// TwinCAT 3 PLC project HL3
// Title: High level object TwinCAT 3 library
// Company: Tomas Rompotl
// ProjectVersion: 0.0.1
// ProgramVersion: 3.1.4023.0
// libraries:
//   Tc2_Standard, * (Beckhoff Automation GmbH)
//   Tc2_System, * (Beckhoff Automation GmbH)
//   Tc2_Utilities, * (Beckhoff Automation GmbH)
//   Tc3_Module, * (Beckhoff Automation GmbH)
//   Base Interfaces,newest,System
// project tree:
//   DataProcessing/Comparison/ CompareAnyType.TcPOU, ComparisonTest.TcPOU, IsGreaterThanOrEqualAnyType.TcPOU, IsNotEqualAnyType.TcPOU, IsLessThanOrEqualAnyType.TcPOU, IsLessThanAnyType.TcPOU, IsEqualAnyType.TcPOU, E_Compare.TcDUT, IsGreaterThanAnyType.TcPOU
//   DataProcessing/QuickSort/ Partition.TcPOU, QuickSort.TcPOU, QuickSortTest.TcPOU
//   DataProcessing/Sort/ E_Order.TcTLEO, SortTest.TcPOU, ST_TestStruct.TcDUT, ST_TestStruct2.TcDUT, _Partition.TcPOU, _QuickSort.TcPOU, Sort.TcPOU
//   General/ E_GeneralResult.TcDUT, E_GeneralStatus.TcTLEO, NegateGeneralResult.TcPOU, Swap.TcPOU, SwapByAddr.TcPOU
//   Lists/ListOfINT/ ListOfINT.TcPOU, ListOfINTTest.TcPOU, NodeINT.TcDUT
//   Lists/List/ List.TcPOU, ListTest.TcPOU, Node.TcDUT
//   Lists/WrappableList/ExampleWithUserDatatype/ WrappableListExample.TcPOU, ListOfUserDatatype.TcPOU, UserDatatype.TcDUT
//   Lists/WrappableList/ WrappableList.TcPOU
//   Misc/ GetAnyType.TcPOU
//   / PlcTask.TcTTO
//   POUs/ MAIN.TcPOU
//   Stringify/ AnyTypeToWSTRING.TcPOU, AnyTypeToSTRING.TcPOU, Stringify.TcPOU
// real-time tasks:
//   TASK PlcTask: cycle T#10ms, priority 20, ADS port 350

CONFIGURATION HL3
    RESOURCE PLC ON TwinCAT3
        TASK PlcTask(INTERVAL := T#10ms, PRIORITY := 20);
        PROGRAM MAIN WITH PlcTask : MAIN;
    END_RESOURCE
END_CONFIGURATION

// ---- DataProcessing/Comparison/E_Compare.TcDUT

{attribute 'qualified_only'}
{attribute 'strict'}
TYPE E_Compare :
(
	EQUAL,
	NOT_EQUAL,
	LESS_THAN,
	LOWER_THAN_OR_EQUAL,
	GREATER_THAN,
	GREATER_THAN_OR_EQUAL
);
END_TYPE

// ---- DataProcessing/Sort/E_Order.TcTLEO

{attribute 'qualified_only'}
{attribute 'strict'}
TYPE E_Order :
(
	ASCENDING,
	DESCENDING
);
END_TYPE

// ---- DataProcessing/Sort/ST_TestStruct.TcDUT
TYPE ST_TestStruct :
STRUCT
	by_this	: ST_TestStruct2;
END_STRUCT
END_TYPE

// ---- DataProcessing/Sort/ST_TestStruct2.TcDUT
TYPE ST_TestStruct2 :
STRUCT
	nested_variable : TIME;
END_STRUCT
END_TYPE

// ---- General/E_GeneralResult.TcDUT

{attribute 'qualified_only'}
{attribute 'strict'}
TYPE E_GeneralResult :
(
	NONE := 0,
	OK,
	NOK,
	_TRUE, // TRUE is keyword
	_FALSE // FALSE is keyword
	
);
END_TYPE

// ---- General/E_GeneralStatus.TcTLEO

{attribute 'qualified_only'}
{attribute 'strict'}
TYPE E_GeneralStatus :
(
	NONE := 0,
	STOP,
	BUSY,
	DONE,
	ERROR,
	INPUT_ERROR,
	INTERRUPT
);
END_TYPE

// ---- Lists/ListOfINT/NodeINT.TcDUT
{attribute 'enable_dynamic_creation'}
TYPE NodeINT :
STRUCT
	data : INT;
	next : POINTER TO NodeINT;
END_STRUCT
END_TYPE

// ---- Lists/List/Node.TcDUT

{attribute 'enable_dynamic_creation'}
TYPE Node :
STRUCT
	data : POINTER TO BYTE;
	next : POINTER TO Node;
END_STRUCT
END_TYPE

// ---- Lists/WrappableList/ExampleWithUserDatatype/UserDatatype.TcDUT
TYPE UserDatatype :
STRUCT
	VarBOOL : BOOL;
	VarREAL : REAL;
	VarARRAYINT : ARRAY[0..9] OF INT;
END_STRUCT
END_TYPE

// ---- POUs/MAIN.TcPOU

PROGRAM MAIN
VAR
	a : ARRAY[0..5] OF REAL;
	b : ARRAY[10..15] OF REAL;
END_VAR


ListOfINTTest();
ListTest();
WrappableListExample();

QuickSortTest();
SortTest();
ComparisonTest();

END_PROGRAM

// ---- Lists/ListOfINT/ListOfINTTest.TcPOU
PROGRAM ListOfINTTest
VAR
	listOfINTExample : ListOfINT;
	
	// init
	first : BOOL := TRUE;
	reinit : BOOL;
	
	// insert test
	insertTest : BOOL;
	insertNumber : INT := 42;
	insertIndex : INT := 0;
	
	// remove test
	removeTest : BOOL;
	removeIndex : INT := 0;
	
	// prepend test
	prependTest : BOOL;
	prependData : INT := -10;
	
	// removeAll test
	removeAllTest : BOOL;
	
	// debug
	test : ARRAY[0..30] OF INT;
	
	// hokusy pokusy
	info : __SYSTEM.VAR_INFO;
	
END_VAR

IF first THEN
	first := FALSE;
	listOfINTExample.Append(3);
	listOfINTExample.Append(4);
	listOfINTExample.Append(5).Prepend(2).Prepend(1);
END_IF;
IF reinit THEN
	reinit := FALSE;
	listOfINTExample.FB_init(FALSE, FALSE);
	first := TRUE;
END_IF

IF insertTest THEN
	insertTest := FALSE;
	listOfINTExample.Insert(insertIndex, insertNumber);
END_IF
IF removeTest THEN
	removeTest := FALSE;
	listOfINTExample.Remove(removeIndex);
END_IF
IF removeAllTest THEN
	removeAllTest := FALSE;
	listOfINTExample.RemoveAll();
END_IF


info := __VARINFO(listOfINTExample);
test[0] := listOfINTExample.Get(0);
test[1] := listOfINTExample.Get(1);
test[2] := listOfINTExample.Get(2);
test[3] := listOfINTExample.Get(3);
test[4] := listOfINTExample.Get(4);
test[5] := listOfINTExample.Get(5);
test[6] := listOfINTExample.Get(6);
test[7] := listOfINTExample.Get(7);
test[8] := listOfINTExample.Get(8);
test[9] := listOfINTExample.Get(9);

test[20] := listOfINTExample.Get(-1);
test[21] := listOfINTExample.Get(-2);
test[22] := listOfINTExample.Get(-3);
test[23] := listOfINTExample.Get(-4);
test[24] := listOfINTExample.Get(-5);
test[25] := listOfINTExample.Get(-6);
test[26] := listOfINTExample.Get(-7);
test[27] := listOfINTExample.Get(-8);
test[28] := listOfINTExample.Get(-9);
test[29] := listOfINTExample.Get(-10);

listOfINTExample.count;

END_PROGRAM

// ---- Lists/ListOfINT/ListOfINT.TcPOU

FUNCTION_BLOCK ListOfINT
VAR_INPUT
END_VAR
VAR_OUTPUT
	count : UINT;
END_VAR
VAR
	head : POINTER TO NodeINT := NULL;
	tail : POINTER TO NodeINT := NULL;
END_VAR


// linked list implementation reference:
// https://www.codesdope.com/blog/article/c-linked-lists-in-c-singly-linked-list/


METHOD Append : REFERENCE TO ListOfINT
VAR_INPUT
	data : INT;
END_VAR
VAR
	new : POINTER TO NodeINT;
END_VAR

Append REF= THIS^;

new := __NEW(NodeINT);
new^.data := data;
new^.next := NULL;

IF head = NULL THEN
	head := new;
	tail := new;
ELSE
	tail^.next := new;
	tail := tail^.next;
END_IF
count := count + 1;
END_METHOD


METHOD Get : INT
VAR_INPUT
	// indexing from end allowed
	// index = 0 returns first element
	// index = 1 returns seconds element
	// index = -1 returns last element
	// index = -2 return before-last element
	index : INT;
END_VAR
VAR
	current : POINTER TO NodeINT := NULL;
	getIndex : INT;
	i : INT;
END_VAR

IF head = NULL THEN
	Get := 0;
	RETURN;
END_IF;

// Calculate actual index in List
getIndex := (count * BOOL_TO_INT(index < 0)) + index;

// Return 0 for invalid indexes
IF 	(getIndex >= count) OR	// Indexing from begin begins with 0
	(getIndex < 0) // Indexing from end begins with -1
THEN
	Get := 0;
	RETURN;
END_IF


current := head;
FOR i := 1 TO getIndex DO // we already got head in previous line, that's why it's from 1
	IF current^.next = NULL THEN
		Get := 0; RETURN;
	END_IF
	current := current^.next;
END_FOR
Get := current^.data;
END_METHOD

// Inserts new element into given index. Negative indexing is supported
METHOD Insert : REFERENCE TO ListOfINT
VAR_INPUT
	(*
		0 = Prepend;
		1 = Insert into second position;
		-2 = Insert into second position from end;
		-1 = Append;
	*)
	index : INT;
	data : INT;
END_VAR
VAR
	new : POINTER TO NodeINT;
	current : POINTER TO NodeINT;
	insertIndex : INT;
	i : INT;
END_VAR

Insert REF= THIS^;

new := __NEW(NodeINT);
new^.data := data;

// Calculate actual index in List
insertIndex := ((count + 1) * BOOL_TO_INT(index < 0)) + index;

IF insertIndex >= count // Index too high -> append to end
THEN
	Append(data);
	RETURN;
ELSIF insertIndex <= 0 // Index too high from the end -> prepend to beginning
THEN
	Prepend(data);
	RETURN;
END_IF

current := head;
FOR i := 1 TO insertIndex - 1 DO
	current := current^.next;
END_FOR
new^.next := current^.next;
current^.next := new;
count := count + 1;
END_METHOD


METHOD IsEmpty : BOOL
VAR_INPUT
END_VAR

IsEmpty := head = NULL;
END_METHOD


// Pushes data to the beginning of the list
METHOD Prepend : REFERENCE TO ListOfINT
VAR_INPUT
	data : INT;
END_VAR
VAR
	new : POINTER TO NodeINT;
END_VAR

Prepend REF= THIS^;

new := __NEW(NodeINT);
new^.data := data;
new^.next := head;

IF head = NULL THEN
	head := new;
	tail := new;
ELSE
	head := new;
END_IF
count := count + 1;
END_METHOD


METHOD Remove : REFERENCE TO ListOfINT;
VAR_INPUT
	index : INT;
END_VAR
VAR
	current : POINTER TO NodeINT := NULL;
	removeIndex : INT;	
	nodeToRemove : POINTER TO NodeINT;
	i : INT;
END_VAR

Remove REF= THIS^;

IF head = NULL THEN
	RETURN;
END_IF;

// Calculate actual index in List
removeIndex := (count * BOOL_TO_INT(index < 0)) + index; 

// Cancel removal for invalid indexes
IF 	(removeIndex >= count) OR // Indexing from begin begins with 0
	(removeIndex < 0) // Indexing from end begins with -1
THEN
	RETURN;
END_IF

IF removeIndex = 0 THEN
	nodeToRemove := head;
	head := head^.next;
ELSE
	current := head;
	FOR i := 1 TO removeIndex - 1 DO
		current := current^.next;
	END_FOR
	nodeToRemove := current^.next;
	current^.next := current^.next^.next;
END_IF
IF nodeToRemove = tail THEN
	tail := current;
END_IF
__DELETE(nodeToRemove);
count := count - 1;
END_METHOD


METHOD RemoveAll : REFERENCE TO ListOfINT
VAR_INPUT
END_VAR

WHILE head <> NULL DO
	Remove(0);
END_WHILE
END_METHOD

END_FUNCTION_BLOCK

// ---- Lists/List/ListTest.TcPOU

PROGRAM ListTest
VAR
	//testing
	testList : List;
	testVar	: REAL;
	appendTest : BOOL := TRUE;
	getTest : BOOL := TRUE;
	removeTest : BOOL;
	getVar : ARRAY[0..19] OF REAL;
	
END_VAR


IF appendTest THEN
	appendTest := FALSE;
	testVar := 1;
	testList.Append(testVar);
	testVar := 2;
	testList.Append(testVar);
	testVar := 3.14;
	testList.Append(testVar);
	testVar := -2;
	testList.Prepend(testVar);
	testVar := -3;
	testList.Prepend(testVar);
	testVar := -1;
	testList.Insert(2, testVar);
	testVar := 3;
	testList.Insert(5, testVar);
END_IF
IF getTest THEN
//	getTest := FALSE;
	ClearTestReadArray();
	testList.Get(0, getVar[0]);
	testList.Get(1, getVar[1]);
	testList.Get(2, getVar[2]);
	testList.Get(3, getVar[3]);
	testList.Get(4, getVar[4]);
	testList.Get(5, getVar[5]);
	testList.Get(6, getVar[6]);
	testList.Get(7, getVar[7]);
	testList.Get(8, getVar[8]);
	
	testList.Get(-1, getVar[10]);
	testList.Get(-2, getVar[11]);
	testList.Get(-3, getVar[12]);
	testList.Get(-4, getVar[13]);
	testList.Get(-5, getVar[14]);
	testList.Get(-6, getVar[15]);
	testList.Get(-7, getVar[16]);
	testList.Get(-8, getVar[17]);
END_IF
IF removeTest THEN
	removeTest := FALSE;
	testList.Remove(1);
END_IF

METHOD ClearTestReadArray : BOOL
VAR
	i : INT;
END_VAR
FOR i := 0 TO 19 DO
	getVar[i] := 0;
END_FOR
END_METHOD

END_PROGRAM

// ---- Lists/List/List.TcPOU

FUNCTION_BLOCK List
VAR_INPUT
END_VAR
VAR_OUTPUT
	count : UINT;
	_typeClass : __SYSTEM.TYPE_CLASS; // Type of data object - primitives or Userdef
	_classSize : DINT; // Size of data object - useful to check type of Userdef typeclass
END_VAR
VAR
	head : POINTER TO Node := NULL;
	tail : POINTER TO Node := NULL;
END_VAR


METHOD Append : REFERENCE TO List
VAR_INPUT
	data : ANY;
END_VAR
VAR
	new : POINTER TO Node;
END_VAR

Append REF= THIS^;

IF NOT IsTypeClassCorrect(data) THEN
	RETURN;
END_IF
SetTypeClass(data);

new := __NEW(Node);
new^.data := __NEW(BYTE, classSize);
MEMCPY(new^.data, data.pValue, classSize);
new^.next := NULL;

IF head = NULL THEN
	head := new;
	tail := new;
ELSE
	tail^.next := new;
	tail := tail^.next;
END_IF
count := count + 1;
END_METHOD


//{attribute 'monitoring' := 'call'}
// Size of data object - useful to check type of Userdef typeclass
PROPERTY classSize : DINT
GET

classSize := _classSize;
END_GET
SET // PRIVATE

_classSize := classSize;
END_SET
END_PROPERTY


METHOD Get : REFERENCE TO List
VAR_INPUT
	// indexing from end allowed
	// index = 0 returns first element
	// index = 1 returns seconds element
	// index = -1 returns last element
	// index = -2 return before-last element
	index : INT;
	destinationVariable : ANY;
END_VAR
VAR
	current : POINTER TO Node := NULL;
	getIndex : INT;
	i : INT;
END_VAR

IF NOT IsTypeClassCorrect(destinationVariable) THEN
	RETURN;
END_IF;

IF head = NULL THEN
	RETURN;
END_IF;

// Calculate actual index in List
getIndex := (count * BOOL_TO_INT(index < 0)) + index;

// Return 0 for invalid indexes
IF 	(getIndex >= count) OR	// Indexing from begin begins with 0
	(getIndex < 0) // Indexing from end begins with -1
THEN
	RETURN;
END_IF


current := head;
FOR i := 1 TO getIndex DO // we already got head in previous line, that's why it's from 1
	IF current^.next = NULL THEN
		RETURN;
	END_IF
	current := current^.next;
END_FOR
MEMMOVE(destinationVariable.pValue, current^.data, classSize);
END_METHOD

// Inserts new element into given index. Negative indexing is supported
METHOD Insert : REFERENCE TO List
VAR_INPUT
	(*
		0 = Prepend;
		1 = Insert into second position;
		-2 = Insert into second position from end;
		-1 = Append;
	*)
	index : INT;
	data : ANY;
END_VAR
VAR
	new : POINTER TO Node;
	current : POINTER TO Node;
	insertIndex : INT;
	i : INT;
END_VAR

Insert REF= THIS^;

IF NOT IsTypeClassCorrect(data) THEN
	RETURN;
END_IF
SetTypeClass(data);

new := __NEW(Node);
new^.data := __NEW(BYTE, classSize);
MEMCPY(new^.data, data.pValue, classSize);

// Calculate actual index in List
insertIndex := ((count + 1) * BOOL_TO_INT(index < 0)) + index;

IF insertIndex >= count // Index too high -> append to end
THEN
	Append(data);
	RETURN;
ELSIF insertIndex <= 0 // Index too high from the end -> prepend to beginning
THEN
	Prepend(data);
	RETURN;
END_IF

current := head;
FOR i := 1 TO insertIndex - 1 DO
	current := current^.next;
END_FOR
new^.next := current^.next;
current^.next := new;
count := count + 1;
END_METHOD


METHOD IsEmpty : BOOL
VAR_INPUT
END_VAR

IsEmpty := head = NULL;
END_METHOD


METHOD IsTypeClassCorrect : BOOL
VAR_INPUT
	CheckedVariable : ANY;
END_VAR

IF classSize = 0 THEN
	IsTypeClassCorrect := TRUE;
	RETURN;
END_IF
IsTypeClassCorrect := typeClass = CheckedVariable.TypeClass AND classSize = CheckedVariable.diSize;
END_METHOD


// Pushes data to the beginning of the list
METHOD Prepend : REFERENCE TO List
VAR_INPUT
	data : ANY;
END_VAR
VAR
	new : POINTER TO Node;
END_VAR

Prepend REF= THIS^;

IF NOT IsTypeClassCorrect(data) THEN
	RETURN;
END_IF
SetTypeClass(data);

new := __NEW(Node);
new^.data := __NEW(BYTE, classSize);
MEMCPY(new^.data, data.pValue, classSize);
new^.next := head;

IF head = NULL THEN
	head := new;
	tail := new;
ELSE
	head := new;
END_IF
count := count + 1;
END_METHOD


METHOD Remove : REFERENCE TO List;
VAR_INPUT
	index : INT;
END_VAR
VAR
	current : POINTER TO Node := NULL;
	removeIndex : INT;	
	nodeToRemove : POINTER TO Node;
	i : INT;
END_VAR

Remove REF= THIS^;

IF head = NULL THEN
	RETURN;
END_IF;

// Calculate actual index in List
removeIndex := (count * BOOL_TO_INT(index < 0)) + index; 

// Cancel removal for invalid indexes
IF 	(removeIndex >= count) OR // Indexing from begin begins with 0
	(removeIndex < 0) // Indexing from end begins with -1
THEN
	RETURN;
END_IF

IF removeIndex = 0 THEN
	nodeToRemove := head;
	head := head^.next;
ELSE
	current := head;
	FOR i := 1 TO removeIndex - 1 DO
		current := current^.next;
	END_FOR
	nodeToRemove := current^.next;
	current^.next := current^.next^.next;
END_IF
IF nodeToRemove = tail THEN
	tail := current;
END_IF
__DELETE(nodeToRemove^.data);
__DELETE(nodeToRemove);
count := count - 1;
END_METHOD


METHOD RemoveAll : REFERENCE TO List
VAR_INPUT
END_VAR

WHILE head <> NULL DO
	Remove(0);
END_WHILE
END_METHOD


METHOD SetTypeClass : BOOL
VAR_INPUT
	ReferenceVariable : ANY; // Pass any variable of your chosen type. It will only be used to obtain data type
END_VAR

IF classSize = 0 THEN
	typeClass := ReferenceVariable.TypeClass;
	classSize := ReferenceVariable.diSize;
	SetTypeClass := TRUE;
END_IF
END_METHOD


//{attribute 'monitoring' := 'call'}
// Type of data object - primitives or Userdef
PROPERTY typeClass : __SYSTEM.TYPE_CLASS
GET

typeClass := _typeClass;
END_GET
SET // PRIVATE

_typeClass := typeClass;
END_SET
END_PROPERTY

END_FUNCTION_BLOCK

// ---- Lists/WrappableList/ExampleWithUserDatatype/WrappableListExample.TcPOU
PROGRAM WrappableListExample
VAR
	myList	: ListOfUserDatatype;
	
	data1 : UserDatatype;
	data2 : UserDatatype;
	
	dataRead : UserDatatype;
	boolRead : BOOL;
	boolTest : BOOL;
	append : BOOL := TRUE;
	
	
END_VAR

IF append THEN
	data1.VarBOOL := TRUE;
	data1.VarREAL := 3.14;
	data1.VarARRAYINT[0] := 1;
	data1.VarARRAYINT[1] := 2;
	data1.VarARRAYINT[2] := 4;
	data1.VarARRAYINT[3] := -8;
	data1.VarARRAYINT[4] := -16;
	
	data2.VarBOOL := FALSE;
	data2.VarREAL := 1.618;
	data2.VarARRAYINT[0] := -555;
	data2.VarARRAYINT[1] := 123;
	data2.VarARRAYINT[2] := -10;
	data2.VarARRAYINT[3] := -0;
	data2.VarARRAYINT[4] := -18;

	append := FALSE;
	myList.Append(data1).Append(data2);
END_IF

myList.Get(0);

boolRead := myList.Get(0).VarBOOL;
myList.Get(0).VarREAL;

dataRead := myList.Get(1);

END_PROGRAM

// ---- Lists/WrappableList/ExampleWithUserDatatype/ListOfUserDatatype.TcPOU
FUNCTION_BLOCK ListOfUserDatatype EXTENDS WrappableList
VAR_INPUT
END_VAR
VAR_OUTPUT
END_VAR
VAR
END_VAR

METHOD Append : REFERENCE TO ListOfUserDatatype
VAR_INPUT
	data : UserDatatype;
END_VAR
Append REF= THIS^;
SUPER^._Append(data);
END_METHOD


METHOD Get : REFERENCE TO UserDatatype
VAR_INPUT
	index : INT;
END_VAR
VAR
	value : UserDatatype;
END_VAR

_Get(index, value);
Get REF= value;
END_METHOD

END_FUNCTION_BLOCK

// ---- Lists/WrappableList/WrappableList.TcPOU

FUNCTION_BLOCK WrappableList
VAR_INPUT
END_VAR
VAR_OUTPUT
	count : UINT;
	_typeClass : __SYSTEM.TYPE_CLASS; // Type of data object - primitives or Userdef
	_classSize : DINT; // Size of data object - useful to check type of Userdef typeclass
END_VAR
VAR
	head : POINTER TO Node := NULL;
	tail : POINTER TO Node := NULL;
END_VAR

METHOD PROTECTED _Append : REFERENCE TO WrappableList
VAR_INPUT
	data : ANY;
END_VAR
VAR
	new : POINTER TO Node;
END_VAR
_Append REF= THIS^;

IF NOT IsTypeClassCorrect(data) THEN
	RETURN;
END_IF
SetTypeClass(data);

new := __NEW(Node);
new^.data := __NEW(BYTE, classSize);
MEMCPY(new^.data, data.pValue, classSize);
new^.next := NULL;

IF head = NULL THEN
	head := new;
	tail := new;
ELSE
	tail^.next := new;
	tail := tail^.next;
END_IF
count := count + 1;
END_METHOD


METHOD PROTECTED _Get : REFERENCE TO WrappableList
VAR_INPUT
	// indexing from end allowed
	// index = 0 returns first element
	// index = 1 returns seconds element
	// index = -1 returns last element
	// index = -2 return before-last element
	index : INT;
	destinationVariable : ANY;
END_VAR
VAR
	current : POINTER TO Node := NULL;
	getIndex : INT;
	i : INT;
END_VAR

IF NOT IsTypeClassCorrect(destinationVariable) THEN
	RETURN;
END_IF;

IF head = NULL THEN
	RETURN;
END_IF;

// Calculate actual index in List
getIndex := (count * BOOL_TO_INT(index < 0)) + index;

// Return 0 for invalid indexes
IF 	(getIndex >= count) OR	// Indexing from begin begins with 0
	(getIndex < 0) // Indexing from end begins with -1
THEN
	RETURN;
END_IF


current := head;
FOR i := 1 TO getIndex DO // we already got head in previous line, that's why it's from 1
	IF current^.next = NULL THEN
		RETURN;
	END_IF
	current := current^.next;
END_FOR
MEMMOVE(destinationVariable.pValue, current^.data, classSize);
END_METHOD


//{attribute 'monitoring' := 'call'}
// Size of data object - useful to check type of Userdef typeclass
PROPERTY classSize : DINT
GET

classSize := _classSize;
END_GET
SET // PRIVATE

_classSize := classSize;
END_SET
END_PROPERTY

// Inserts new element into given index. Negative indexing is supported
METHOD Insert : REFERENCE TO WrappableList
VAR_INPUT
	(*
		0 = Prepend;
		1 = Insert into second position;
		-2 = Insert into second position from end;
		-1 = Append;
	*)
	index : INT;
	data : ANY;
END_VAR
VAR
	new : POINTER TO Node;
	current : POINTER TO Node;
	insertIndex : INT;
	i : INT;
END_VAR

Insert REF= THIS^;

IF NOT IsTypeClassCorrect(data) THEN
	RETURN;
END_IF
SetTypeClass(data);

new := __NEW(Node);
new^.data := __NEW(BYTE, classSize);
MEMCPY(new^.data, data.pValue, classSize);

// Calculate actual index in List
insertIndex := ((count + 1) * BOOL_TO_INT(index < 0)) + index;

IF insertIndex >= count // Index too high -> append to end
THEN
	_Append(data);
	RETURN;
ELSIF insertIndex <= 0 // Index too high from the end -> prepend to beginning
THEN
	Prepend(data);
	RETURN;
END_IF

current := head;
FOR i := 1 TO insertIndex - 1 DO
	current := current^.next;
END_FOR
new^.next := current^.next;
current^.next := new;
count := count + 1;
END_METHOD


METHOD IsEmpty : BOOL
VAR_INPUT
END_VAR

IsEmpty := head = NULL;
END_METHOD


METHOD IsTypeClassCorrect : BOOL
VAR_INPUT
	CheckedVariable : ANY;
END_VAR

IF classSize = 0 THEN
	IsTypeClassCorrect := TRUE;
	RETURN;
END_IF
IsTypeClassCorrect := typeClass = CheckedVariable.TypeClass AND classSize = CheckedVariable.diSize;
END_METHOD


// Pushes data to the beginning of the list
METHOD Prepend : REFERENCE TO WrappableList
VAR_INPUT
	data : ANY;
END_VAR
VAR
	new : POINTER TO Node;
END_VAR

Prepend REF= THIS^;

IF NOT IsTypeClassCorrect(data) THEN
	RETURN;
END_IF
SetTypeClass(data);

new := __NEW(Node);
new^.data := __NEW(BYTE, classSize);
MEMCPY(new^.data, data.pValue, classSize);
new^.next := head;

IF head = NULL THEN
	head := new;
	tail := new;
ELSE
	head := new;
END_IF
count := count + 1;
END_METHOD


METHOD Remove : REFERENCE TO WrappableList;
VAR_INPUT
	index : INT;
END_VAR
VAR
	current : POINTER TO Node := NULL;
	removeIndex : INT;	
	nodeToRemove : POINTER TO Node;
	i : INT;
END_VAR

Remove REF= THIS^;

IF head = NULL THEN
	RETURN;
END_IF;

// Calculate actual index in List
removeIndex := (count * BOOL_TO_INT(index < 0)) + index; 

// Cancel removal for invalid indexes
IF 	(removeIndex >= count) OR // Indexing from begin begins with 0
	(removeIndex < 0) // Indexing from end begins with -1
THEN
	RETURN;
END_IF

IF removeIndex = 0 THEN
	nodeToRemove := head;
	head := head^.next;
ELSE
	current := head;
	FOR i := 1 TO removeIndex - 1 DO
		current := current^.next;
	END_FOR
	nodeToRemove := current^.next;
	current^.next := current^.next^.next;
END_IF
IF nodeToRemove = tail THEN
	tail := current;
END_IF
__DELETE(nodeToRemove^.data);
__DELETE(nodeToRemove);
count := count - 1;
END_METHOD


METHOD RemoveAll : REFERENCE TO WrappableList
VAR_INPUT
END_VAR

WHILE head <> NULL DO
	Remove(0);
END_WHILE
END_METHOD


METHOD SetTypeClass : BOOL
VAR_INPUT
	ReferenceVariable : ANY; // Pass any variable of your chosen type. It will only be used to obtain data type
END_VAR

IF classSize = 0 THEN
	typeClass := ReferenceVariable.TypeClass;
	classSize := ReferenceVariable.diSize;
	SetTypeClass := TRUE;
END_IF
END_METHOD


//{attribute 'monitoring' := 'call'}
// Type of data object - primitives or Userdef
PROPERTY typeClass : __SYSTEM.TYPE_CLASS
GET

typeClass := _typeClass;
END_GET
SET // PRIVATE

_typeClass := typeClass;
END_SET
END_PROPERTY

END_FUNCTION_BLOCK

// ---- DataProcessing/QuickSort/QuickSortTest.TcPOU

PROGRAM QuickSortTest
VAR
	TestArray0 : ARRAY[0..20] OF REAL := [
		1, 2, 3, 4, 5, 6, 7, 8, 9, 10,
		42, 3.14, 0.618, 1.618, 2.618
	];
	TestArray1 : ARRAY[0..1] OF REAL := [0.1, -0.2];
	
	init : BOOL;
	sort : BOOL;
END_VAR


IF init THEN
	init := FALSE;
	reinit();
END_IF

IF sort THEN
	sort := FALSE;
	QuickSort(TestArray0, 0, 20);
	QuickSort(TestArray1, 0, 1);
END_IF


METHOD reinit : BOOL
VAR_INPUT
END_VAR
VAR CONSTANT
	Array0 : ARRAY[0..20] OF REAL := [
		1, 2, 3, 4, 5, 6, 7, 8, 9, 10,
		42, 3.14, 0.618, 1.618, 2.618
	];
	Array1 : ARRAY[0..1] OF REAL := [0.1, -0.2];
END_VAR

TestArray0 := Array0;
TestArray1 := Array1;
END_METHOD

END_PROGRAM

// ---- DataProcessing/Sort/Sort.TcPOU

// sort any array of anything
FUNCTION Sort : E_GeneralStatus
VAR_INPUT
	Arr 			: ANY; // data to be sorted, get size of array
	FirstElement 	: ANY; // get size of element to be able to get count of elements and iterate over them
	SortBy 			: ANY; // possibility to pass array of structures and sort by some of its member - this will get its type and offset in element. Will have its own function SortBy() later
	Order 			: E_Order;
END_VAR
VAR
	ElemSize		: DINT;
	ElemCount 		: DINT;
	MemberOffset 	: DWORD;
	
	StartIndex 		: DINT := 0;
	EndIndex 		: DINT;
END_VAR


IF 	arr.pValue = 0 OR firstElement.pValue = 0 OR sortBy.pValue = 0 OR 
	arr.diSize = 0 OR firstElement.diSize = 0 OR sortBy.pValue = 0 THEN

	Sort := E_GeneralStatus.INPUT_ERROR;
	RETURN;
END_IF

elemCount := arr.diSize / firstElement.diSize;
memberOffset := sortBy.pValue - firstElement.pValue;
EndIndex := ElemCount - 1;

_QuickSort(Arr, FirstElement, SortBy, MemberOffset, StartIndex, EndIndex, Order);

END_FUNCTION

// ---- DataProcessing/Sort/_QuickSort.TcPOU

FUNCTION _QuickSort
VAR_INPUT
	Arr					: __SYSTEM.AnyType;
	FirstElement		: __SYSTEM.AnyType;
	SortBy				: __SYSTEM.AnyType;
	MemberOffset		: DWORD;
	StartIndex			: DINT; // Start index
	EndIndex			: DINT; // End index
	Order 				: E_Order;
END_VAR
VAR 
	PivotIndex			: DINT; // Partitioning point
END_VAR


IF StartIndex < EndIndex THEN

	PivotIndex := _Partition(Arr, FirstElement, SortBy, MemberOffset, StartIndex, EndIndex, Order);
	_QuickSort(Arr, FirstElement, SortBy, MemberOffset, StartIndex, PivotIndex - 1, Order);
	_QuickSort(Arr, FirstElement, SortBy, MemberOffset, PivotIndex + 1, EndIndex, Order);
END_IF

END_FUNCTION

// ---- DataProcessing/Sort/_Partition.TcPOU

// Function used in QuickSort
FUNCTION _Partition : DINT
VAR_INPUT
	Arr					: __SYSTEM.AnyType;
	FirstElement		: __SYSTEM.AnyType;
	SortBy				: __SYSTEM.AnyType;
	MemberOffset		: DWORD;
	StartIndex			: DINT; // Starting comparision index
	EndIndex			: DINT; // Ending comparision index
	Order 				: E_Order;
END_VAR
VAR
	Pivot				: POINTER TO BYTE; // Compared number
	Leftwall			: DINT; // New pivot location
	Iterator			: DINT; // For iterator variable
	IterAdr				: POINTER TO BYTE;
	compA				: __SYSTEM.AnyType := SortBy; // get data of compared variable
	compB				: __SYSTEM.AnyType := SortBy;
END_VAR


Pivot := Arr.pValue + FirstElement.diSize * EndIndex;

Leftwall := StartIndex;

FOR Iterator := StartIndex TO EndIndex - 1 DO

	IterAdr := Arr.pValue + FirstElement.diSize * Iterator;
	
	compA.pValue := IterAdr + MemberOffset; // data of compared variable stays the same, just point to other value
	compB.pValue := Pivot + MemberOffset;
	
	CASE Order OF
		E_Order.ASCENDING:
			IF IsLessThanOrEqualAnyType(compA, compB) = E_GeneralResult._TRUE THEN

				SwapByAddr(IterAdr, Arr.pValue + FirstElement.diSize * Leftwall, FirstElement.diSize);
				Leftwall := Leftwall + 1;
			END_IF
		E_Order.DESCENDING:
			IF IsGreaterThanOrEqualAnyType(compA, compB) = E_GeneralResult._TRUE THEN

				SwapByAddr(IterAdr, Arr.pValue + FirstElement.diSize * Leftwall, FirstElement.diSize);
				Leftwall := Leftwall + 1;
			END_IF
	END_CASE
END_FOR

SwapByAddr(Arr.pValue + FirstElement.diSize * Leftwall, Pivot, FirstElement.diSize);

_Partition := Leftwall;

END_FUNCTION

// ---- DataProcessing/Comparison/IsLessThanOrEqualAnyType.TcPOU
FUNCTION IsLessThanOrEqualAnyType : E_GeneralResult
VAR_INPUT
	A					: __SYSTEM.AnyType; // A and B have to be same type
	B					: __SYSTEM.AnyType; // A and B have to be same type
END_VAR

IsLessThanOrEqualAnyType := NegateGeneralResult(IsGreaterthanAnyType(A, B));

END_FUNCTION

// ---- General/NegateGeneralResult.TcPOU

FUNCTION NegateGeneralResult : E_GeneralResult
VAR_INPUT
	result		: E_GeneralResult;
END_VAR
VAR
END_VAR


CASE result OF
	E_GeneralResult.OK:
		NegateGeneralResult := E_GeneralResult.NOK;
	E_GeneralResult.NOK:
		NegateGeneralResult := E_GeneralResult.OK;
	E_GeneralResult._TRUE:
		NegateGeneralResult := E_GeneralResult._FALSE;
	E_GeneralResult._FALSE:
		NegateGeneralResult := E_GeneralResult._TRUE;
	ELSE
		NegateGeneralResult := result;
END_CASE

END_FUNCTION

// ---- DataProcessing/Comparison/IsGreaterThanAnyType.TcPOU

FUNCTION IsGreaterThanAnyType : E_GeneralResult
VAR_INPUT
	A					: __SYSTEM.AnyType; // A and B have to be same type
	B					: __SYSTEM.AnyType; // A and B have to be same type
END_VAR
VAR
	isGreaterThan			: BOOL;
END_VAR


IF A.TypeClass <> B.TypeClass THEN

	RETURN;
END_IF

CASE UDINT_TO_INT(A.TypeClass) OF
    IBaseLibrary.TypeClass.TYPE_BOOL :
        isGreaterThan := PBOOL_TO_BOOL(a.pValue) > PBOOL_TO_BOOL(b.pValue);
    IBaseLibrary.TypeClass.TYPE_BIT :
        isGreaterThan := BYTE_TO_BIT(a.pValue^) > BYTE_TO_BIT(b.pValue^);
    IBaseLibrary.TypeClass.TYPE_BYTE :
        isGreaterThan := a.pValue^ > b.pValue^;
    IBaseLibrary.TypeClass.TYPE_WORD :
        isGreaterThan := PWORD_TO_WORD(a.pValue) > PWORD_TO_WORD(b.pValue);
    IBaseLibrary.TypeClass.TYPE_DWORD :
        isGreaterThan := PDWORD_TO_DWORD(a.pValue) > PDWORD_TO_DWORD(b.pValue);
    IBaseLibrary.TypeClass.TYPE_LWORD :
        isGreaterThan := PLWORD_TO_LWORD(a.pValue) > PLWORD_TO_LWORD(b.pValue);
    IBaseLibrary.TypeClass.TYPE_SINT :
        isGreaterThan := PSINT_TO_SINT(a.pValue) > PSINT_TO_SINT(b.pValue);
    IBaseLibrary.TypeClass.TYPE_INT :
        isGreaterThan := PINT_TO_INT(a.pValue) > PINT_TO_INT(b.pValue);
    IBaseLibrary.TypeClass.TYPE_DINT :
        isGreaterThan := PDINT_TO_DINT(a.pValue) > PDINT_TO_DINT(b.pValue);
    IBaseLibrary.TypeClass.TYPE_LINT :
        isGreaterThan := PLINT_TO_LINT(a.pValue) > PLINT_TO_LINT(b.pValue);
    IBaseLibrary.TypeClass.TYPE_USINT :
        isGreaterThan := PUSINT_TO_USINT(a.pValue) > PUSINT_TO_USINT(b.pValue);
    IBaseLibrary.TypeClass.TYPE_UINT :
        isGreaterThan := PUINT_TO_UINT(a.pValue) > PUINT_TO_UINT(b.pValue);
    IBaseLibrary.TypeClass.TYPE_UDINT :
        isGreaterThan := PUDINT_TO_UDINT(a.pValue) > PUDINT_TO_UDINT(b.pValue);
    IBaseLibrary.TypeClass.TYPE_ULINT :
        isGreaterThan := PULINT_TO_ULINT(a.pValue) > PULINT_TO_ULINT(b.pValue);
    IBaseLibrary.TypeClass.TYPE_REAL :
        isGreaterThan := PREAL_TO_REAL(a.pValue) > PREAL_TO_REAL(b.pValue);
    IBaseLibrary.TypeClass.TYPE_LREAL :
        isGreaterThan := PLREAL_TO_LREAL(a.pValue) > PLREAL_TO_LREAL(b.pValue);
    IBaseLibrary.TypeClass.TYPE_STRING :
        isGreaterThan := PSTRING_TO_STRING(a.pValue) > PSTRING_TO_STRING(b.pValue);
    IBaseLibrary.TypeClass.TYPE_TIME :
        isGreaterThan := PTIME_TO_TIME(a.pValue) > PTIME_TO_TIME(b.pValue);
    IBaseLibrary.TypeClass.TYPE_DATE :
        isGreaterThan := PDATE_TO_DATE(a.pValue) > PDATE_TO_DATE(b.pValue);
    IBaseLibrary.TypeClass.TYPE_DATEANDTIME :
        isGreaterThan := PDT_TO_DT(a.pValue) > PDT_TO_DT(b.pValue);
    IBaseLibrary.TypeClass.TYPE_TIMEOFDAY :
        isGreaterThan := PTOD_TO_TOD(a.pValue) > PTOD_TO_TOD(b.pValue);
    IBaseLibrary.TypeClass.TYPE_POINTER :
        isGreaterThan := a.pValue > b.pValue;
    IBaseLibrary.TypeClass.TYPE_LTIME :
        isGreaterThan := PLTIME_TO_LTIME(a.pValue) > PLTIME_TO_LTIME(b.pValue);
	ELSE
		RETURN;
END_CASE

IF isGreaterThan THEN

	IsGreaterThanAnyType := E_GeneralResult._TRUE;
ELSE

	IsGreaterThanAnyType := E_GeneralResult._FALSE;
END_IF

END_FUNCTION

// ---- General/SwapByAddr.TcPOU

// Swaps values of to variables
FUNCTION SwapByAddr : E_GeneralStatus
VAR_INPUT
	A : POINTER TO BYTE;
	B : POINTER TO BYTE;
	Length : DINT;
END_VAR
VAR
	Temp : POINTER TO BYTE;
END_VAR


IF A = 0 OR B = 0 THEN
	
	SwapByAddr := E_GeneralStatus.INPUT_ERROR;
	RETURN;
END_IF

Temp := __NEW(BYTE, Length);

MEMCPY(Temp, A, Length);
MEMCPY(A, B, Length);
MEMCPY(B, Temp, Length);

__DELETE(Temp);

SwapByAddr := E_GeneralStatus.DONE;

END_FUNCTION

// ---- DataProcessing/Comparison/IsGreaterThanOrEqualAnyType.TcPOU
FUNCTION IsGreaterThanOrEqualAnyType : E_GeneralResult
VAR_INPUT
	A					: __SYSTEM.AnyType; // A and B have to be same type
	B					: __SYSTEM.AnyType; // A and B have to be same type
END_VAR

IsGreaterThanOrEqualAnyType := NegateGeneralResult(IsLessThanAnyType(A, B));

END_FUNCTION

// ---- DataProcessing/Comparison/IsLessThanAnyType.TcPOU
FUNCTION IsLessThanAnyType : E_GeneralResult
VAR_INPUT
	A					: __SYSTEM.AnyType; // A and B have to be same type
	B					: __SYSTEM.AnyType; // A and B have to be same type
END_VAR
VAR
	isLessThan			: BOOL;
END_VAR

IF A.TypeClass <> B.TypeClass THEN

	RETURN;
END_IF

CASE UDINT_TO_INT(A.TypeClass) OF
    IBaseLibrary.TypeClass.TYPE_BOOL :
        isLessThan := PBOOL_TO_BOOL(a.pValue) < PBOOL_TO_BOOL(b.pValue);
    IBaseLibrary.TypeClass.TYPE_BIT :
        isLessThan := BYTE_TO_BIT(a.pValue^) < BYTE_TO_BIT(b.pValue^);
    IBaseLibrary.TypeClass.TYPE_BYTE :
        isLessThan := a.pValue^ < b.pValue^;
    IBaseLibrary.TypeClass.TYPE_WORD :
        isLessThan := PWORD_TO_WORD(a.pValue) < PWORD_TO_WORD(b.pValue);
    IBaseLibrary.TypeClass.TYPE_DWORD :
        isLessThan := PDWORD_TO_DWORD(a.pValue) < PDWORD_TO_DWORD(b.pValue);
    IBaseLibrary.TypeClass.TYPE_LWORD :
        isLessThan := PLWORD_TO_LWORD(a.pValue) < PLWORD_TO_LWORD(b.pValue);
    IBaseLibrary.TypeClass.TYPE_SINT :
        isLessThan := PSINT_TO_SINT(a.pValue) < PSINT_TO_SINT(b.pValue);
    IBaseLibrary.TypeClass.TYPE_INT :
        isLessThan := PINT_TO_INT(a.pValue) < PINT_TO_INT(b.pValue);
    IBaseLibrary.TypeClass.TYPE_DINT :
        isLessThan := PDINT_TO_DINT(a.pValue) < PDINT_TO_DINT(b.pValue);
    IBaseLibrary.TypeClass.TYPE_LINT :
        isLessThan := PLINT_TO_LINT(a.pValue) < PLINT_TO_LINT(b.pValue);
    IBaseLibrary.TypeClass.TYPE_USINT :
        isLessThan := PUSINT_TO_USINT(a.pValue) < PUSINT_TO_USINT(b.pValue);
    IBaseLibrary.TypeClass.TYPE_UINT :
        isLessThan := PUINT_TO_UINT(a.pValue) < PUINT_TO_UINT(b.pValue);
    IBaseLibrary.TypeClass.TYPE_UDINT :
        isLessThan := PUDINT_TO_UDINT(a.pValue) < PUDINT_TO_UDINT(b.pValue);
    IBaseLibrary.TypeClass.TYPE_ULINT :
        isLessThan := PULINT_TO_ULINT(a.pValue) < PULINT_TO_ULINT(b.pValue);
    IBaseLibrary.TypeClass.TYPE_REAL :
        isLessThan := PREAL_TO_REAL(a.pValue) < PREAL_TO_REAL(b.pValue);
    IBaseLibrary.TypeClass.TYPE_LREAL :
        isLessThan := PLREAL_TO_LREAL(a.pValue) < PLREAL_TO_LREAL(b.pValue);
    IBaseLibrary.TypeClass.TYPE_STRING :
        isLessThan := PSTRING_TO_STRING(a.pValue) < PSTRING_TO_STRING(b.pValue);
    IBaseLibrary.TypeClass.TYPE_TIME :
        isLessThan := PTIME_TO_TIME(a.pValue) < PTIME_TO_TIME(b.pValue);
    IBaseLibrary.TypeClass.TYPE_DATE :
        isLessThan := PDATE_TO_DATE(a.pValue) < PDATE_TO_DATE(b.pValue);
    IBaseLibrary.TypeClass.TYPE_DATEANDTIME :
        isLessThan := PDT_TO_DT(a.pValue) < PDT_TO_DT(b.pValue);
    IBaseLibrary.TypeClass.TYPE_TIMEOFDAY :
        isLessThan := PTOD_TO_TOD(a.pValue) < PTOD_TO_TOD(b.pValue);
    IBaseLibrary.TypeClass.TYPE_POINTER :
        isLessThan := a.pValue < b.pValue;
    IBaseLibrary.TypeClass.TYPE_LTIME :
        isLessThan := PLTIME_TO_LTIME(a.pValue) < PLTIME_TO_LTIME(b.pValue);
	ELSE
		RETURN;
END_CASE

IF isLessThan THEN

	IsLessThanAnyType := E_GeneralResult._TRUE;
ELSE

	IsLessThanAnyType := E_GeneralResult._FALSE;
END_IF

END_FUNCTION

// ---- DataProcessing/QuickSort/QuickSort.TcPOU

// Will sort array of REAL using QuickSort algorithm
FUNCTION QuickSort
VAR_IN_OUT
	ArrayOfREALToSort	: ARRAY[*] OF REAL; // Array to sort
END_VAR
VAR_INPUT
	FirstIndex			: INT; // Start index
	LastIndex			: INT; // End index
END_VAR
VAR 
	PivotLocation		: INT; // Partitioning point
END_VAR


IF FirstIndex < LastIndex THEN
	PivotLocation := Partition(ArrayOfREALToSort, FirstIndex, LastIndex);
	QuickSort(ArrayOfREALToSort, FirstIndex, PivotLocation - 1);
	QuickSort(ArrayOfREALToSort, PivotLocation + 1, LastIndex);
END_IF

END_FUNCTION

// ---- DataProcessing/QuickSort/Partition.TcPOU

// Function used in QuickSort
FUNCTION Partition : INT
VAR_IN_OUT
	ArrayOfREAL			: ARRAY[*] OF REAL; // Partition this array from index nLow to index nHigh
END_VAR
VAR_INPUT
	FirstIndex			: INT; // Starting comparision index
	LastIndex			: INT; // Ending comparision index
END_VAR
VAR
	Pivot				: REAL; // Compared number
	Leftwall			: INT; // New pivot location
	Iterator			: INT; // For iterator variable
END_VAR


Pivot := ArrayOfREAL[LastIndex];
Leftwall := FirstIndex;

FOR Iterator := FirstIndex TO LastIndex - 1 DO
	IF ArrayOfREAL[Iterator] <= Pivot THEN
		Swap(ArrayOfREAL[Iterator], ArrayOfREAL[Leftwall]);
		Leftwall := Leftwall + 1;
	END_IF
END_FOR

Swap(ArrayOfREAL[Leftwall], ArrayOfREAL[LastIndex]);

Partition := Leftwall;

END_FUNCTION

// ---- General/Swap.TcPOU

// Swaps values of to variables
FUNCTION Swap : E_GeneralStatus
VAR_INPUT
	A : ANY;
	B : ANY;
END_VAR
VAR
	Temp : POINTER TO BYTE;
END_VAR


IF a.pValue = 0 OR b.pValue = 0 OR a.diSize <> b.diSize THEN
	
	Swap := E_GeneralStatus.INPUT_ERROR;
	RETURN;
END_IF

Temp := __NEW(BYTE, A.diSize);

MEMCPY(Temp, A.pValue, A.diSize);
MEMCPY(A.pValue, B.pValue, A.diSize);
MEMCPY(B.pValue, Temp, A.diSize);

__DELETE(Temp);

Swap := E_GeneralStatus.DONE;

END_FUNCTION

// ---- DataProcessing/Sort/SortTest.TcPOU

PROGRAM SortTest
VAR
	TestArray0 : ARRAY[0..20] OF REAL := [
		1, 2, 3, 4, 5, 6, 7, 8, 9, 10,
		42, 3.14, 0.618, 1.618, 2.618
	];
	TestArray1 : ARRAY[0..3] OF STRING := ['aaa', 'g', 'aab', 'a'];
	
	sort_array : ARRAY[0..3] OF ST_TestStruct;	// TestArray2
	
	init : BOOL := TRUE;
	startSort : BOOL;
	
	order	: E_Order;
END_VAR


IF init THEN

	init := FALSE;

	reinit();
END_IF

IF startSort THEN

	startSort := FALSE;

	Sort(TestArray0, TestArray0[0], TestArray0[0], order);
	Sort(TestArray1, TestArray1[0], TestArray1[0], order);

	Sort(sort_array, sort_array[0], sort_array[0].by_this.nested_variable, order);
END_IF


METHOD reinit : BOOL
VAR_INPUT
END_VAR
VAR CONSTANT
	Array0 : ARRAY[0..20] OF REAL := [
		1, 2, 3, 4, 5, 6, 7, 8, 9, 10,
		42, 3.14, 0.618, 1.618, 2.618
	];
	Array1 : ARRAY[0..3] OF STRING := ['aaa', 'g', 'aab', 'a'];
END_VAR

TestArray0 := Array0;
TestArray1 := Array1;

sort_array[0].by_this.nested_variable := T#5S;
sort_array[1].by_this.nested_variable := T#1S;
sort_array[2].by_this.nested_variable := T#18D;
sort_array[3].by_this.nested_variable := T#42MS;
END_METHOD

END_PROGRAM

// ---- DataProcessing/Comparison/ComparisonTest.TcPOU
PROGRAM ComparisonTest
VAR
	r1 : LREAL := 3.14;
	r2 : LREAL := -129;
	s1 : STRING := 'towel';
	s2 : STRING := 'galaxy';
	
	at1 : __SYSTEM.AnyType;
	at2 : __SYSTEM.AnyType;
	
	res_r : ARRAY[0..6] OF E_GeneralResult;
	res_s : ARRAY[0..6] OF E_GeneralResult;
	
	test : BOOL;
	
	
	
END_VAR

IF test THEN

	test := FALSE;

	at1 := GetAnyType(r1);
	at2 := GetAnyType(r2);
	
	res_r[0] := IsEqualAnyType(at1, at2);
	res_r[1] := IsNotEqualAnyType(at1, at2);
	res_r[2] := IsLessThanAnyType(at1, at2);
	res_r[3] := IsLessThanOrEqualAnyType(at1, at2);
	res_r[4] := IsGreaterThanAnyType(at1, at2);
	res_r[5] := IsGreaterThanOrEqualAnyType(at1, at2);
	res_r[6] := CompareAnyType(at1, is := E_Compare.GREATER_THAN_OR_EQUAL, at2);

	at1 := GetAnyType(s1);
	at2 := GetAnyType(s2);
	
	res_s[0] := IsEqualAnyType(at1, at2);
	res_s[1] := IsNotEqualAnyType(at1, at2);
	res_s[2] := IsLessThanAnyType(at1, at2);
	res_s[3] := IsLessThanOrEqualAnyType(at1, at2);
	res_s[4] := IsGreaterThanAnyType(at1, at2);
	res_s[5] := IsGreaterThanOrEqualAnyType(at1, at2);
	res_s[6] := CompareAnyType(at1, is := E_Compare.GREATER_THAN_OR_EQUAL, at2);
END_IF

END_PROGRAM

// ---- Misc/GetAnyType.TcPOU
FUNCTION GetAnyType : __SYSTEM.AnyType
VAR_INPUT
	a		: ANY;
END_VAR
VAR
END_VAR

GetAnyType := a;

END_FUNCTION

// ---- DataProcessing/Comparison/IsEqualAnyType.TcPOU

FUNCTION IsEqualAnyType : E_GeneralResult
VAR_INPUT
	A					: __SYSTEM.AnyType; // A and B have to be same type
	B					: __SYSTEM.AnyType; // A and B have to be same type
END_VAR
VAR
	isEqual				: BOOL;
END_VAR


IF A.TypeClass <> B.TypeClass THEN

	RETURN;
END_IF

isEqual := MEMCMP(A.pValue, B.pValue, A.diSize) = 0;

IF isEqual THEN

	IsEqualAnyType := E_GeneralResult._TRUE;
ELSE

	IsEqualAnyType := E_GeneralResult._FALSE;
END_IF

END_FUNCTION

// ---- DataProcessing/Comparison/IsNotEqualAnyType.TcPOU
FUNCTION IsNotEqualAnyType : E_GeneralResult
VAR_INPUT
	A					: __SYSTEM.AnyType; // A and B have to be same type
	B					: __SYSTEM.AnyType; // A and B have to be same type
END_VAR

IsNotEqualAnyType := NegateGeneralResult(IsEqualAnyType(A, B));

END_FUNCTION

// ---- DataProcessing/Comparison/CompareAnyType.TcPOU

FUNCTION CompareAnyType : E_GeneralResult
VAR_INPUT
	A					: __SYSTEM.AnyType; // A and B have to be same type
	is					: E_Compare;
	B					: __SYSTEM.AnyType; // A and B have to be same type
END_VAR
VAR
END_VAR


CASE is OF
	E_Compare.EQUAL:
		CompareAnyType := IsEqualAnyType(A, B);
	E_Compare.NOT_EQUAL:
		CompareAnyType := IsNotEqualAnyType(A, B);
	E_Compare.LESS_THAN:
		CompareAnyType := IsLessThanAnyType(A, B);
	E_Compare.LOWER_THAN_OR_EQUAL:
		CompareAnyType := IsLessThanOrEqualAnyType(A, B);
	E_Compare.GREATER_THAN:
		CompareAnyType := IsGreaterThanAnyType(A, B);
	E_Compare.GREATER_THAN_OR_EQUAL:
		CompareAnyType := IsGreaterThanOrEqualAnyType(A, B);
END_CASE

END_FUNCTION

// ---- Stringify/AnyTypeToWSTRING.TcPOU
FUNCTION AnyTypeToWSTRING : WSTRING
VAR_INPUT
	a	: __System.AnyType;
END_VAR
VAR
END_VAR

CASE UDINT_TO_INT(a.TypeClass) OF
    IBaseLibrary.TypeClass.TYPE_BOOL :
        AnyTypeToWSTRING := BOOL_TO_WSTRING(PBOOL_TO_BOOL(a.pValue));
    IBaseLibrary.TypeClass.TYPE_BIT :
        AnyTypeToWSTRING := BIT_TO_WSTRING(BYTE_TO_BIT(a.pValue^));
    IBaseLibrary.TypeClass.TYPE_BYTE :
        AnyTypeToWSTRING := BYTE_TO_WSTRING(a.pValue^);
    IBaseLibrary.TypeClass.TYPE_WORD :
        AnyTypeToWSTRING := WORD_TO_WSTRING(PWORD_TO_WORD(a.pValue));
    IBaseLibrary.TypeClass.TYPE_DWORD :
        AnyTypeToWSTRING := DWORD_TO_WSTRING(PDWORD_TO_DWORD(a.pValue));
    IBaseLibrary.TypeClass.TYPE_LWORD :
        AnyTypeToWSTRING := LWORD_TO_WSTRING(PLWORD_TO_LWORD(a.pValue));
    IBaseLibrary.TypeClass.TYPE_SINT :
        AnyTypeToWSTRING := SINT_TO_WSTRING(PSINT_TO_SINT(a.pValue));
    IBaseLibrary.TypeClass.TYPE_INT :
        AnyTypeToWSTRING := INT_TO_WSTRING(PINT_TO_INT(a.pValue));
    IBaseLibrary.TypeClass.TYPE_DINT :
        AnyTypeToWSTRING := DINT_TO_WSTRING(PDINT_TO_DINT(a.pValue));
    IBaseLibrary.TypeClass.TYPE_LINT :
        AnyTypeToWSTRING := LINT_TO_WSTRING(PLINT_TO_LINT(a.pValue));
    IBaseLibrary.TypeClass.TYPE_USINT :
        AnyTypeToWSTRING := USINT_TO_WSTRING(PUSINT_TO_USINT(a.pValue));
    IBaseLibrary.TypeClass.TYPE_UINT :
        AnyTypeToWSTRING := UINT_TO_WSTRING(PUINT_TO_UINT(a.pValue));
    IBaseLibrary.TypeClass.TYPE_UDINT :
        AnyTypeToWSTRING := UDINT_TO_WSTRING(PUDINT_TO_UDINT(a.pValue));
    IBaseLibrary.TypeClass.TYPE_ULINT :
        AnyTypeToWSTRING := ULINT_TO_WSTRING(PULINT_TO_ULINT(a.pValue));
    IBaseLibrary.TypeClass.TYPE_REAL :
        AnyTypeToWSTRING := REAL_TO_WSTRING(PREAL_TO_REAL(a.pValue));
    IBaseLibrary.TypeClass.TYPE_LREAL :
        AnyTypeToWSTRING := LREAL_TO_WSTRING(PLREAL_TO_LREAL(a.pValue));
    IBaseLibrary.TypeClass.TYPE_STRING :
        AnyTypeToWSTRING := STRING_TO_WSTRING(PSTRING_TO_STRING(a.pValue));
    IBaseLibrary.TypeClass.TYPE_STRING :
        AnyTypeToWSTRING := TIME_TO_WSTRING(PTIME_TO_TIME(a.pValue));
    IBaseLibrary.TypeClass.TYPE_DATE :
        AnyTypeToWSTRING := DATE_TO_WSTRING(PDATE_TO_DATE(a.pValue));
    IBaseLibrary.TypeClass.TYPE_DATEANDTIME :
        AnyTypeToWSTRING := DT_TO_WSTRING(PDT_TO_DT(a.pValue));
    IBaseLibrary.TypeClass.TYPE_TIMEOFDAY :
        AnyTypeToWSTRING := TOD_TO_WSTRING(PTOD_TO_TOD(a.pValue));
    IBaseLibrary.TypeClass.TYPE_POINTER :
        AnyTypeToWSTRING := STRING_TO_WSTRING(PVOID_TO_HEXSTR(a.pValue, SIZEOF(PVOID), FALSE));
    IBaseLibrary.TypeClass.TYPE_LTIME :
        AnyTypeToWSTRING := LTIME_TO_WSTRING(PLTIME_TO_LTIME(a.pValue));
    ELSE
        AnyTypeToWSTRING := "ERROR: UNSUPPORTED DATA TYPE";
END_CASE

END_FUNCTION

// ---- Stringify/AnyTypeToSTRING.TcPOU
FUNCTION AnyTypeToSTRING : T_MaxString
VAR_INPUT
	a	: __System.AnyType;
END_VAR
VAR
END_VAR

CASE UDINT_TO_INT(a.TypeClass) OF
    IBaseLibrary.TypeClass.TYPE_BOOL :
        AnyTypeToSTRING := BOOL_TO_STRING(PBOOL_TO_BOOL(a.pValue));
    IBaseLibrary.TypeClass.TYPE_BIT :
        AnyTypeToSTRING := BIT_TO_STRING(BYTE_TO_BIT(a.pValue^));
    IBaseLibrary.TypeClass.TYPE_BYTE :
        AnyTypeToSTRING := BYTE_TO_STRING(a.pValue^);
    IBaseLibrary.TypeClass.TYPE_WORD :
        AnyTypeToSTRING := WORD_TO_STRING(PWORD_TO_WORD(a.pValue));
    IBaseLibrary.TypeClass.TYPE_DWORD :
        AnyTypeToSTRING := DWORD_TO_STRING(PDWORD_TO_DWORD(a.pValue));
    IBaseLibrary.TypeClass.TYPE_LWORD :
        AnyTypeToSTRING := LWORD_TO_STRING(PLWORD_TO_LWORD(a.pValue));
    IBaseLibrary.TypeClass.TYPE_SINT :
        AnyTypeToSTRING := SINT_TO_STRING(PSINT_TO_SINT(a.pValue));
    IBaseLibrary.TypeClass.TYPE_INT :
        AnyTypeToSTRING := INT_TO_STRING(PINT_TO_INT(a.pValue));
    IBaseLibrary.TypeClass.TYPE_DINT :
        AnyTypeToSTRING := DINT_TO_STRING(PDINT_TO_DINT(a.pValue));
    IBaseLibrary.TypeClass.TYPE_LINT :
        AnyTypeToSTRING := LINT_TO_STRING(PLINT_TO_LINT(a.pValue));
    IBaseLibrary.TypeClass.TYPE_USINT :
        AnyTypeToSTRING := USINT_TO_STRING(PUSINT_TO_USINT(a.pValue));
    IBaseLibrary.TypeClass.TYPE_UINT :
        AnyTypeToSTRING := UINT_TO_STRING(PUINT_TO_UINT(a.pValue));
    IBaseLibrary.TypeClass.TYPE_UDINT :
        AnyTypeToSTRING := UDINT_TO_STRING(PUDINT_TO_UDINT(a.pValue));
    IBaseLibrary.TypeClass.TYPE_ULINT :
        AnyTypeToSTRING := ULINT_TO_STRING(PULINT_TO_ULINT(a.pValue));
    IBaseLibrary.TypeClass.TYPE_REAL :
        AnyTypeToSTRING := REAL_TO_STRING(PREAL_TO_REAL(a.pValue));
    IBaseLibrary.TypeClass.TYPE_LREAL :
        AnyTypeToSTRING := LREAL_TO_STRING(PLREAL_TO_LREAL(a.pValue));
    IBaseLibrary.TypeClass.TYPE_STRING :
        AnyTypeToSTRING := PSTRING_TO_STRING(a.pValue);
    IBaseLibrary.TypeClass.TYPE_STRING :
        AnyTypeToSTRING := TIME_TO_STRING(PTIME_TO_TIME(a.pValue));
    IBaseLibrary.TypeClass.TYPE_DATE :
        AnyTypeToSTRING := DATE_TO_STRING(PDATE_TO_DATE(a.pValue));
    IBaseLibrary.TypeClass.TYPE_DATEANDTIME :
        AnyTypeToSTRING := DT_TO_STRING(PDT_TO_DT(a.pValue));
    IBaseLibrary.TypeClass.TYPE_TIMEOFDAY :
        AnyTypeToSTRING := TOD_TO_STRING(PTOD_TO_TOD(a.pValue));
    IBaseLibrary.TypeClass.TYPE_POINTER :
        AnyTypeToSTRING := PVOID_TO_HEXSTR(a.pValue, SIZEOF(PVOID), FALSE);
    IBaseLibrary.TypeClass.TYPE_LTIME :
        AnyTypeToSTRING := LTIME_TO_STRING(PLTIME_TO_LTIME(a.pValue));
    ELSE
        AnyTypeToSTRING := 'ERROR: UNSUPPORTED DATA TYPE';
END_CASE

END_FUNCTION

// ---- Stringify/Stringify.TcPOU
FUNCTION Stringify : STRING
VAR_INPUT
	info : __SYSTEM.VAR_INFO;
//	another : INT;
END_VAR
VAR
//	info : __SYSTEM.VAR_INFO;
END_VAR

//info := __VARINFO(data);
Stringify := info.Symbol;

END_FUNCTION
